// TIA Portal V20 export
TYPE "LWONIK_typeFromSafetyEstopStatus"
// stored: Access Published
   STRUCT
      MainOpPanel_EMO : Bool;
      UnwinderLeftEMO : Bool;
      CutterEMO : Bool;
      MagazineEMO : Bool;
      ConveyorEMO : Bool;
      PHMI1_EMO : Bool;
      PHMI2_EMO : Bool;
      BA30_EMO : Bool;
      BA40_EMO : Bool;
      BA15_EMO : Bool;
      BA60_EMO : Bool;
   END_STRUCT;
END_TYPE
